INTERFACE ITF_PMLControl

PROPERTY Mode : E_PMLUnitMode
GET
END_GET
END_PROPERTY

PROPERTY ModeCommand : DINT
SET
END_SET
END_PROPERTY

PROPERTY State : E_PMLState
GET
END_GET
END_PROPERTY

PROPERTY StateCommand : E_PMLCommand
SET
END_SET
END_PROPERTY

END_INTERFACE

(* stored: Version 1.1.0.1, ProductVersion 3.1.4024.11
   Itf ITF_PMLControl: Id {0a595185-78e0-4efa-95fb-0ab72c8c824d}
   Property Mode: Id {68aa19f0-a027-4849-bb10-f5584ab8d043}
   Get Get: Id {e4c0be11-49fb-4f99-95fb-f87a759ebdeb}
   Property ModeCommand: Id {11907bf7-f645-420b-85af-3bf0127cd7f1}
   Set Set: Id {0cf2eb2e-aedc-4e54-afcc-be209278627f}
   Property State: Id {43595dac-7213-416e-a39c-be01c96ab13c}
   Get Get: Id {21f6fac7-5f70-4bd9-8ec4-66822702fbf5}
   Property StateCommand: Id {1c454ada-e18d-4933-8772-ef90079bfec6}
   Set Set: Id {3495e55a-b4ad-4161-a7ba-1793fe13d390} *)
